// Device/Application/ProvRoom_All
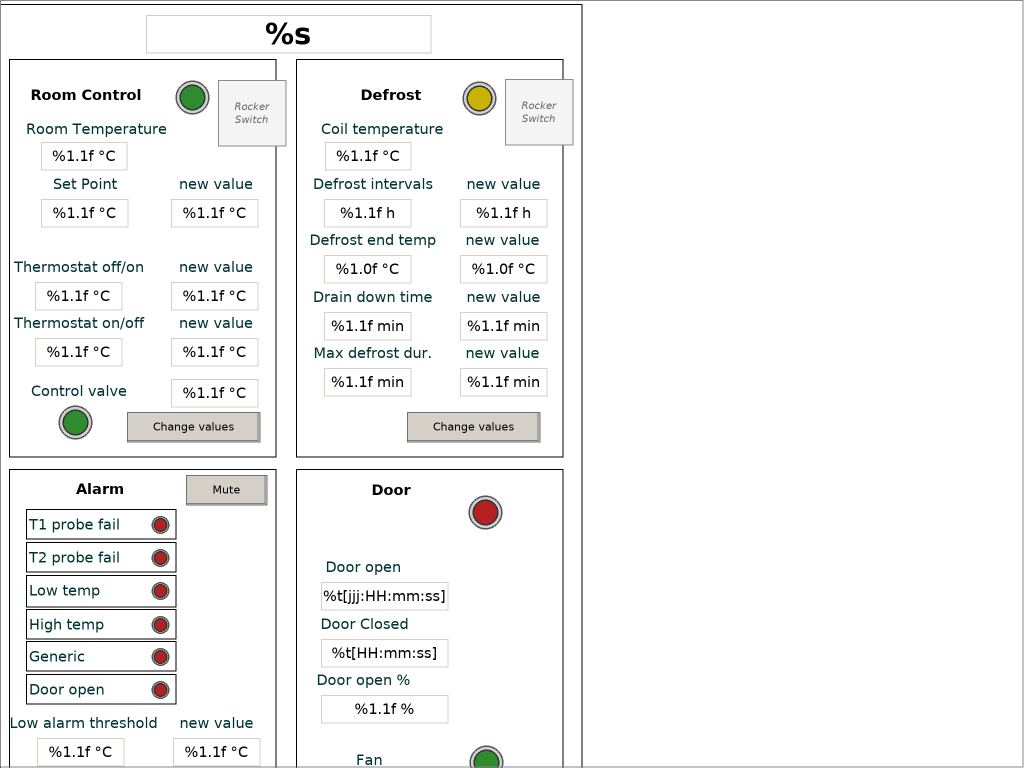
VISUALIZATION ProvRoom_All  // 1024x768
VAR_IN_OUT
	provroomTemp : FB_Provision_room();
END_VAR
    Rectangle (0,4 582x954)
    Rectangle (296,59 267x398), colour toggle: not.Provision_1.control_button
    Rectangle (9,59 267x398), colour toggle: not.Provision_1.control_button
    Lamp1 (533,911 39x39), variable: Provision_1.modbus_communication, style: Lamp-Lamp1-Green
    Textfield (41,199 87x28), "%1.1f °C", text variable: provroomTemp.P_Setpoint
    Label (25,112 143x34), "Room Temperature"
    Textfield (41,142 86x28), "%1.1f °C", tooltip "Provision_1.temp_provision_room", text variable: provroomTemp.P_Room_temp
    Label (15,167 140x34), "Set Point"
    Label (457,913 76x34), "Comms:"
    Label (11,80 150x30), "Room Control"
    Lamp1 (173,78 39x39), variable: provroomTemp.P_Machine_standby, style: Lamp-Lamp1-Green
    Textfield (171,199 87x28), "%1.1f °C", text variable: provroomTemp.P_setpoint_write
        OnMouseClick: write provroomTemp.P_setpoint_write via Edit
    Label (146,167 140x34), "new value"
    Textfield (35,282 87x28), "%1.1f °C", text variable: provroomTemp.P_Thermostat_OFF_ON_ref_to_SP
        p4168582468: provroomTemp.P_Thermostat_OFF_ON_ref_to_SP
    Label (9,250 140x34), "Thermostat off/on"
    Textfield (171,282 87x28), "%1.1f °C", text variable: provroomTemp.P_Thermostat_OFF_ON_ref_to_SP_write
        OnMouseClick: write provroomTemp.P_Thermostat_OFF_ON_ref_to_SP_write via Edit
    Label (146,250 140x34), "new value"
    Textfield (35,338 87x28), "%1.1f °C", text variable: provroomTemp.P_Thermostat_ON_OFF_ref_to_SP
        p4168582468: provroomTemp.P_Thermostat_ON_OFF_ref_to_SP
    Label (9,306 140x34), "Thermostat on/off"
    Textfield (171,338 87x28), "%1.1f °C", text variable: provroomTemp.P_Thermostat_ON_OFF_ref_to_SP_write
        OnMouseClick: write provroomTemp.P_Thermostat_ON_OFF_ref_to_SP_write via Edit
    Label (146,306 140x34), "new value"
    Rectangle (9,469 267x431), colour toggle: not.Provision_1.control_button
    Rectangle (26,509 150x30)
    Rectangle (26,542 150x30)
    Rectangle (26,575 150x32)
    Rectangle (26,609 150x30)
    Label (26,514 105x21), "T1 probe fail"
    Lamp1 (149,515 23x20), tooltip "Provision_1.T1_failure", variable: Provision_1.T1_failure, style: Lamp-Lamp1-Red
    Label (26,547 105x21), "T2 probe fail"
    Lamp1 (149,548 23x20), tooltip "Provision_1.T2_failure", variable: Provision_1.T2_failure, style: Lamp-Lamp1-Red
    Label (26,580 105x21), "Low temp"
    Lamp1 (149,581 23x20), tooltip "Provision_1.Low_temperature", variable: provroomTemp.P_Low_temperature, style: Lamp-Lamp1-Red
    Label (26,614 130x21), "High temp"
    Lamp1 (149,615 23x20), variable: provroomTemp.P_High_temperature, style: Lamp-Lamp1-Red
    Rectangle (26,641 150x30)
    Rectangle (26,674 150x30)
    Label (26,646 105x21), "Generic"
    Lamp1 (149,647 23x20), variable: provroomTemp.P_Generic_alarm, style: Lamp-Lamp1-Red
    Label (26,679 105x21), "Door open"
    Lamp1 (149,680 23x20), tooltip "Provision_1.Door_open_alarm", variable: Provision_1.Door_open_alarm, style: Lamp-Lamp1-Red
    Textfield (37,738 87x28), "%1.1f °C", text variable: provroomTemp.P_Low_temperature_alarm_threshold
    Label (11,706 150x34), "Low alarm threshold"
    Textfield (173,738 87x28), "%1.1f °C", text variable: Provision_1.Low_temperature_alarm_thres_write
        OnMouseClick: write Provision_1.Low_temperature_alarm_thres_write via Default
    Label (173,706 87x34), "new value"
    Textfield (37,794 87x28), "%1.1f °C", text variable: provroomTemp.P_High_temperature_alarm_threshold
    Label (11,762 150x34), "High alarm threshold"
    Textfield (173,794 87x28), "%1.1f °C", text variable: Provision_1.High_temperature_alarm_thres_write
        OnMouseClick: write Provision_1.High_temperature_alarm_thres_write via Default
    Label (171,762 89x34), "new value"
    Button (127,852 133x30), "Change values"
        OnMouseDown:  ToggleVariable=Provision_1.xtrigger_alarm
        OnMouseUp:  ToggleVariable=Provision_1.xtrigger_alarm
    Button (127,412 133x30), "Change values"
        OnMouseDown:  ToggleVariable=provroomTemp.P_xTrigger_setpoint
        OnMouseUp:  ToggleVariable=provroomTemp.P_xTrigger_setpoint
    Button (407,412 133x30), "Change values"
        OnMouseDown:  ToggleVariable=Provision_1.xtrigger_defrost
        OnMouseUp:  ToggleVariable=Provision_1.xtrigger_defrost
    Button (186,475 81x30), "Mute"
        OnMouseDown:  ToggleVariable=Provision_1.xtrigger_mute
        OnMouseUp:  ToggleVariable=Provision_1.xtrigger_mute
    Textfield (324,199 87x28), "%1.1f h", text variable: provroomTemp.P_Time_based_defrost
        p4168582468: provroomTemp.P_Time_based_defrost
    Label (298,167 150x34), "Defrost intervals"
    Textfield (460,199 87x28), "%1.1f h", text variable: Provision_1.Time_based_defrost_write
        p4168582468: Provision_1.Time_based_defrost_write
        OnMouseClick: write the text variable via Default
    Label (460,167 87x34), "new value"
    Textfield (324,255 87x28), "%1.0f °C", text variable: provroomTemp.P_Defrost_end_temperature
        p4168582468: provroomTemp.P_Defrost_end_temperature
    Label (298,223 150x34), "Defrost end temp"
    Textfield (460,255 87x28), "%1.0f °C", text variable: Provision_1.Defrost_end_temperature_write
        p4168582468: Provision_1.Defrost_end_temperature_write
        OnMouseClick: write the text variable via Default
    Label (458,223 89x34), "new value"
    Textfield (324,312 87x28), "%1.1f min", text variable: provroomTemp.P_Drain_down_time
        p4168582468: provroomTemp.P_Drain_down_time
    Label (298,280 150x34), "Drain down time"
    Textfield (460,312 87x28), "%1.1f min", text variable: Provision_1.Drain_down_time_write
        p4168582468: Provision_1.Drain_down_time_write
        OnMouseClick: write the text variable via Edit
    Label (460,280 87x34), "new value"
    Textfield (324,368 87x28), "%1.1f min", text variable: provroomTemp.P_Maximum_defrost_duration
        p4168582468: provroomTemp.P_Maximum_defrost_duration
    Label (298,336 150x34), "Max defrost dur."
    Textfield (460,368 87x28), "%1.1f min", text variable: Provision_1.Maximum_defrost_duration_write
        OnMouseClick: write the text variable via Default
    Label (458,336 89x34), "new value"
    RockerSwitch (505,79 68x66), variable: Provision_1.defrost_button, behaviour: TOGGLE, style: Switch-RockerSwitch-Gray
        OnValueChanged:  ToggleVariable=Provision_1.xtrigger_man_defrost
    Label (316,80 150x30), "Defrost"
    RockerSwitch (218,80 68x66), variable: Provision_1.control_button, behaviour: TOGGLE, style: Switch-RockerSwitch-Gray
        OnValueChanged:  ToggleVariable=Provision_1.xtrigger_control
    Lamp1 (460,79 39x39), variable: provroomTemp.P_Defrost, style: Lamp-Lamp1-Yellow
    Textfield (325,142 86x28), "%1.1f °C", text variable: provroomTemp.P_Temp_defrost
    Label (311,112 143x34), "Coil temperature"
    Rectangle (296,469 267x431), colour toggle: not.Provision_1.control_button
    Button (407,822 133x30), "reset timers", pressed state: Provision_1.resettimer_button
        OnMouseDown:  ToggleVariable=Provision_1.resettimer_button
        OnMouseUp:  ToggleVariable=Provision_1.resettimer_button
    Label (316,475 150x30), "Door"
    Label (25,474 150x30), "Alarm"
    Textfield (321,582 127x28), "%t[jjj:HH:mm:ss]", text variable: Provision_1.opentime_tot
        p4168582468: Provision_1.opentime_tot
        OnMouseClick: write the text variable via Default
    Label (319,550 89x34), "Door open"
    Textfield (321,639 127x28), "%t[HH:mm:ss]", text variable: Provision_1.closetime_tot
        p4168582468: Provision_1.closetime_tot
        OnMouseClick: write the text variable via Default
    Label (321,607 87x34), "Door Closed"
    Textfield (321,695 127x28), "%1.1f %", text variable: Provision_1.opentime_proc
        OnMouseClick: write the text variable via Default
    Label (319,663 89x34), "Door open %"
    Lamp1 (56,403 39x39), variable: provroomTemp.P_Dout3, style: Lamp-Lamp1-Green
    Label (9,374 140x34), "Control valve"
    Lamp1 (466,493 39x39), variable: provroomTemp.P_Door_open, style: Lamp-Lamp1-Red
    Lamp1 (467,743 39x39), variable: provroomTemp.P_Dout2, style: Lamp-Lamp1-Green
    Label (325,743 89x34), "Fan"
    Textfield (146,15 285x38), "%s", text variable: provroomTemp.P_Provision_name
    Textfield (171,379 87x28), "%1.1f °C", text variable: provroomTemp.P_test_input
        OnMouseClick: write Provision_1.setp_write via Default
END_VISUALIZATION

// Device/Application/ProvRoomTemp
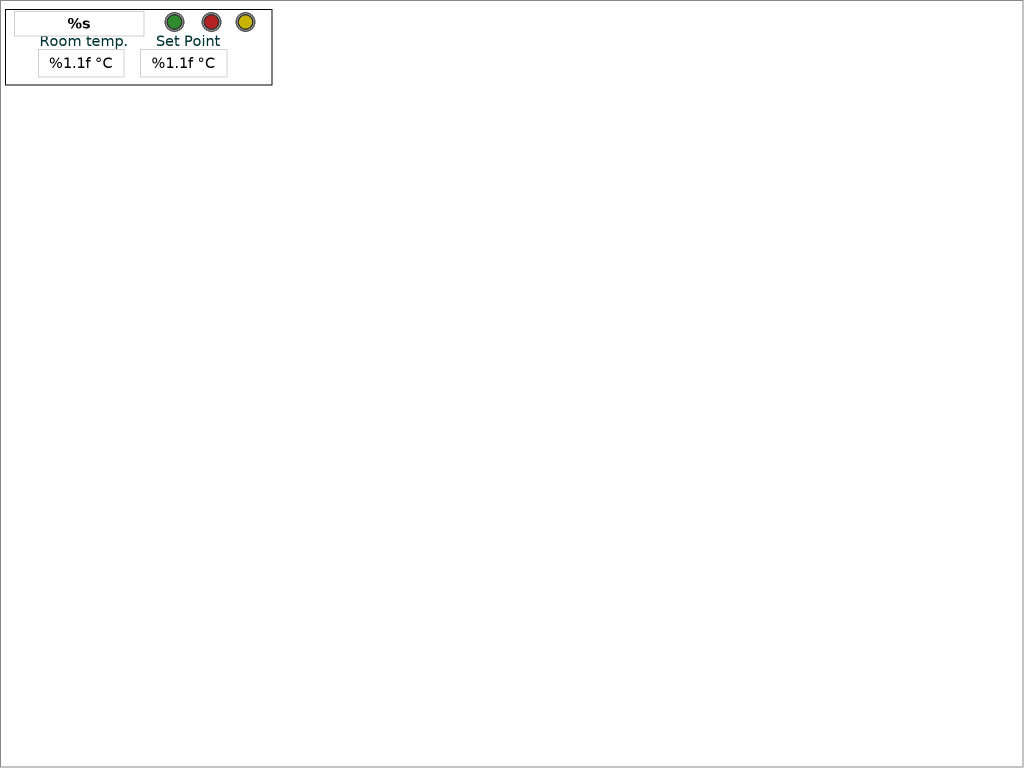
VISUALIZATION ProvRoomTemp  // 1024x768
VAR_IN_OUT
		provroomTemp : FB_Provision_room();
END_VAR
    Rectangle (5,9 267x76), colour toggle: not.Provision_1.control_button
        OnMouseClick:  Assign=Provision_1_2_3_SysOverview, Type=Assignment
    Textfield (140,49 87x28), "%1.1f °C", text variable: provroomTemp.P_Setpoint
    Label (24,24 120x34), "Room temp."
    Textfield (38,49 86x28), "%1.1f °C", text variable: provroomTemp.P_Room_temp
    Label (118,24 140x34), "Set Point"
    Lamp1 (200,10 23x24), variable: provroomTemp.P_Alarm, style: Lamp-Lamp1-Red
    Lamp1 (163,10 23x24), variable: provroomTemp.P_Machine_standby, style: Lamp-Lamp1-Green
    Textfield (14,11 130x25), "%s", text variable: provroomTemp.I_Provision_name
    Lamp1 (234,10 23x24), variable: provroomTemp.P_Alarm, style: Lamp-Lamp1-Yellow
END_VISUALIZATION
